// TIA Portal V16 export
// export: Created 2022-07-21T09:35:15.839518Z, ExportSetting WithDefaults, DisplayName Totally Integrated Automation Portal, DisplayVersion V16 Update 4, DisplayName TIA Portal Version Control Interface, DisplayVersion V16 Update 2, DisplayName TIA Portal Openness, DisplayVersion V16 Update 4, DisplayName SINAMICS Startdrive Advanced, DisplayVersion V16 Update 5, DisplayName SINAMICS Startdrive G130, G150, S120, S150, SINAMICS MV, S210, DisplayVersion V16 Update 5, DisplayName SINAMICS Startdrive G110M, G120, G120C, G120D, G120P, G115D, DisplayVersion V16 Update 5, DisplayName STEP 7 Professional, DisplayVersion V16 Update 4, DisplayName STEP 7 Safety, DisplayVersion V16, DisplayName WinCC Advanced, DisplayVersion V16 Update 4
DATA_BLOCK "LAxisBasics_AxisDataBlock"   // DB810
{ S7_Optimized_Access := 'TRUE' }
AUTHOR : ArSc
FAMILY : LAxisBasics
VERSION : 1.1
// stored: AutoNumber false, DBAccessibleFromOPCUA true, InstanceOfName LAxisBasics_typeAxisDataBlock, InstanceOfType UDT, IsOnlyStoredInLoadMemory false, IsWriteProtectedInAS false
"LAxisBasics_typeAxisDataBlock"
   // VAR RETAIN
   //    axis { S7_SetPoint := 'True'} : Array[0..10] of "LAxisBasics_typeAxisBasicsData";
   // END_VAR
BEGIN
   // axis[0] : PA27205 Gasket układ 2D (S120)
   // axis[1] : PA27205.1 Gasket układ 2D (S120)
   // axis[2] : PA27305 Gasket układ 3D (S120)
   // axis[3] : PA27305.1 Gasket układ 3D (S120)
   // axis[4] : PA27405 Gasket układ 3D (S120)
   // axis[5] : PA27405.1 Gasket układ stacjonarny (S120)
   // axis[6] : PA27505 Podawanie Body (S120)
   // axis[7] : PA27505.1 Podawanie Lid (S120)
   // axis[8] : Rezerwa
   // axis[9] : Rezerwa
   // axis[10] : Rezerwa
   axis[0].axisControl.axisControlCommand.homePosition := 450.0;
   axis[4].axisControl.axisControlCommand.homePosition := 45.0;
END_DATA_BLOCK
